Staubli VAL3: Deplacementpion.pgx

public program Deplacementpion(num x_nPointDepart, num x_nPointArrivee)
begin
  //met à jour position des cases noires
  call CasesNoires()


  //Deplacementpion(X,Y) -> deplacement du pion de X vers Y


  //Deplacement vers le pion en X
  movej( appro(pCaseNoire[x_nPointDepart], trAppro), tTool, mDeplacement)

  //s'approche et prend le pion en X
  close(tTool)
  movel( pCaseNoire[x_nPointDepart], tTool, mPrise)
  open(tTool)

  movel( appro(pCaseNoire[x_nPointDepart], trAppro), tTool, mDeplacement)

  //Deplacement vers Y puis approche vers Y
  movej ( appro(pCaseNoire[x_nPointArrivee], trAppro), tTool, mDeplacement)
  movel( pCaseNoire[x_nPointArrivee], tTool, mPrise)

  //lache la piece et remonte
  close(tTool)
  movel( appro(pCaseNoire[x_nPointArrivee], trAppro), tTool, mDeplacement)


end
